// TIA Portal project "1_Basic_PID_Control" (V19)

(* hardware
DEVICE "S7-1500/ET200MP station_1"  S7-1500 station
   slot 0: "Rail_0"  Rack  6ES7 590-1***0-0AA0
   slot 1: "PLC_1"  CPU 1513-1 PN  6ES7 513-1AL02-0AB0  V2.9
      slot 3: "CPU display_1"  6ES7591-1AA00-0AA0
      slot 32768: "PROFINET interface_1"  X1
         slot 32769: "Port_1"  X1 P1
         slot 32770: "Port_2"  X1 P2
      slot 34817: "Virtual CP interface port_1"  Virtual CP interface port  Virtual CP interface port
*)

// ===== PLC "PLC_1"  CPU 1513-1 PN =====

VAR_GLOBAL   // PLC tag table "Default tag table"
   "LV Output" AT %MD0 : Real;
   "SP Output" AT %MD4 : Real;
   "Error" AT %MD8 : Real;
   "FV Output" AT %MD12 : Real;
   "FV Buffer" AT %MD16 : Real;
END_VAR

VAR_GLOBAL   // PLC tag table "Tag table from XML_1"
   "Start_PB" AT %I0.0 : Bool;
   "Reset_PB" AT %I0.1 : Bool;
   "Stop_PB" AT %I0.2 : Bool;
   "FACTORY I/O (Running)" AT %I0.3 : Bool;
   "Start light" AT %Q0.0 : Bool;
   "Reset light" AT %Q0.1 : Bool;
   "Stop light" AT %Q0.2 : Bool;
   "Level meter" AT %ID30 : Real;
   "Flow meter" AT %ID34 : Real;
   "Setpoint" AT %ID38 : Real;
   "Fill valve" AT %QD30 : Real;
   "Discharge valve" AT %QD34 : Real;
   "SP" AT %QD38 : DInt;
   "PV" AT %QD42 : DInt;
END_VAR

ORGANIZATION_BLOCK "Main"   // OB1, LAD, ProgramCycle
TITLE = "Main Program Sweep (Cycle)"
{ S7_Optimized_Access := 'TRUE' }
VERSION : 0.1
   VAR_INPUT
      Initial_Call : Bool;   // Initial call of this OB
      Remanence : Bool;   // =True, if remanent data are available
   END_VAR
BEGIN

REGION Network 2: Level Meter
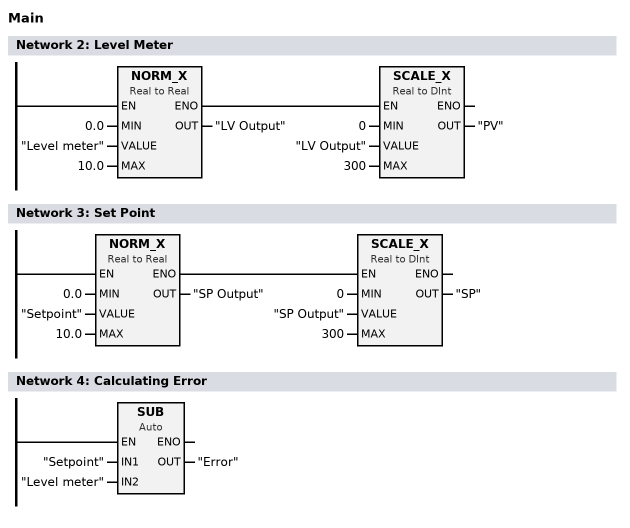
   RUNG wire#powerrail
      { S7_Templates := "[SrcType := Real, DestType := Real]" } Normalize(min := 0.0, value := "Level meter", max := 10.0, out => "LV Output")
      { S7_Templates := "[SrcType := Real, DestType := DInt]" } Scale(min := 0, value := "LV Output", max := 300, out => "PV")
   END_RUNG
   // the same network as SCL:
   "LV Output" := NORM_X(MIN := 0.0, VALUE := "Level meter", MAX := 10.0);
   "PV" := SCALE_X(MIN := 0, VALUE := "LV Output", MAX := 300);
END_REGION

REGION Network 3: Set Point
   RUNG wire#powerrail
      { S7_Templates := "[SrcType := Real, DestType := Real]" } Normalize(min := 0.0, value := "Setpoint", max := 10.0, out => "SP Output")
      { S7_Templates := "[SrcType := Real, DestType := DInt]" } Scale(min := 0, value := "SP Output", max := 300, out => "SP")
   END_RUNG
   // the same network as SCL:
   "SP Output" := NORM_X(MIN := 0.0, VALUE := "Setpoint", MAX := 10.0);
   "SP" := SCALE_X(MIN := 0, VALUE := "SP Output", MAX := 300);
END_REGION

REGION Network 4: Calculating Error
   RUNG wire#powerrail
      Sub(in1 := "Setpoint", in2 := "Level meter", out => "Error")
   END_RUNG
   // the same network as SCL:
   "Error" := "Setpoint" - "Level meter";
END_REGION
END_ORGANIZATION_BLOCK

ORGANIZATION_BLOCK "CyclicInterrupt"   // OB30, LAD, CyclicInterrupt
{ S7_Optimized_Access := 'TRUE' }
VERSION : 0.1
   VAR_INPUT
      Initial_Call : Bool;   // Initial call of this OB
      Event_Count : Int;   // Events discarded
   END_VAR
BEGIN

REGION Network 1
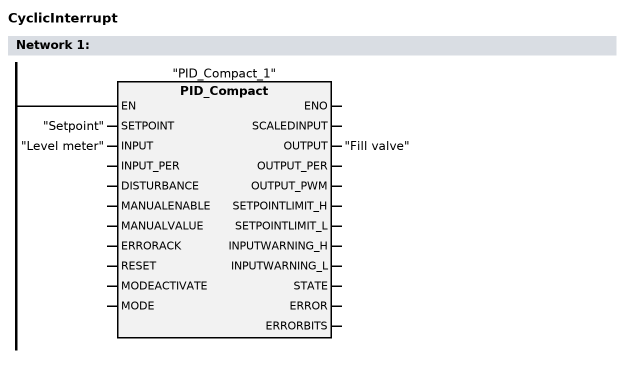
   "PID_Compact_1"(Setpoint := "Setpoint", Input := "Level meter", Output => "Fill valve");   // PID_Compact
END_REGION
END_ORGANIZATION_BLOCK